// TwinCAT 3 PLC project Types
// Title: Types
// Company: TomasRompotl
// ProjectVersion: 0.0.2
// ProgramVersion: 3.1.4024.0
// libraries:
//   Tc2_Standard, * (Beckhoff Automation GmbH)
//   Tc2_System, * (Beckhoff Automation GmbH)
//   Tc2_Utilities, * (Beckhoff Automation GmbH)
//   Tc3_JsonXml, * (Beckhoff Automation GmbH)
//   Tc3_Module, * (Beckhoff Automation GmbH)
//   Base Interfaces,newest,System
// project tree:
//   Any/ AnyTypeUnion.TcDUT, ToAnyType.TcPOU, IsAnyTypeBinded.TcPOU
//   Binding/ BoolBindingReadOnly.TcPOU, BoolBindable.TcIO (not stored), NotBind.TcPOU (not stored), Bind.TcPOU (not stored)
//   Disposable/ Disposable.TcIO
//   Numbers/ Integer.TcDUT (not stored), Decimal.TcDUT, Positive.TcDUT
//   Queryable/ Queryable.TcIO (not stored)
//   Reflection/ Reflection.TcPOU
//   Values/BooleanExpression/ BooleanOperator.TcDUT (not stored), BooleanExpression.TcPOU
//   Values/BooleanExpression/Functions/ And2.TcPOU, And3.TcPOU (not stored), And4.TcPOU, Or2.TcPOU (not stored), Or3.TcPOU, Or4.TcPOU (not stored), Xor2.TcPOU, Xor3.TcPOU (not stored), Xor4.TcPOU (not stored)
//   Values/ BoolValues.TcGVL (not stored), FalseBoolValue.TcPOU, TrueBoolValue.TcPOU (not stored), BoolValue.TcIO
//   Version/ Global_Version.TcGVL
// real-time tasks:
//   TASK BindingTestTask: cycle T#10ms, priority 20, ADS port 350
//   TASK PlcTask: cycle T#10ms, priority 21, ADS port 351
//   TASK PlcTask1: cycle T#10ms, priority 22, ADS port 352
//   TASK PlcTask2: cycle T#10ms, priority 23, ADS port 353

// ---- Any/AnyTypeUnion.TcDUT
TYPE AnyTypeUnion :
UNION
	BOOL_ : BOOL;
	BIT_ : BIT;
	BYTE_ : BYTE;
	WORD_ : WORD;
	DWORD_ : DWORD;
	LWORD_ : LWORD;
	SINT_ : SINT;
	INT_ : INT;
	DINT_ : DINT;
	LINT_ : LINT;
	USINT_ : USINT;
	UINT_ : UINT;
	UDINT_ : UDINT;
	ULINT_ : ULINT;
	REAL_ : REAL;
	LREAL_ : LREAL;
	STRING_ : T_MaxString;
	TIME_ : TIME;
	DATE_ : DATE;
	DATEANDTIME_ : DATE_AND_TIME;
	TIMEOFDAY_ : TIME_OF_DAY;
	POINTER_ : POINTER TO BYTE;
	LTIME_ : LTIME;
END_UNION
END_TYPE

// ---- Numbers/Decimal.TcDUT
TYPE Decimal : LREAL; END_TYPE

// ---- Numbers/Positive.TcDUT
TYPE Positive : ULINT; END_TYPE

// ---- Version/Global_Version.TcGVL
{attribute 'TcGenerated'}
{attribute 'no-analysis'}
{attribute 'linkalways'}
// This function has been automatically generated from the project information.
VAR_GLOBAL CONSTANT
	{attribute 'const_non_replaced'}
	stLibVersion_Types : ST_LibVersion := (iMajor := 0, iMinor := 0, iBuild := 2, iRevision := 0, nFlags := 0, sVersion := '0.0.2');
END_VAR

// ---- Disposable/Disposable.TcIO
INTERFACE Disposable EXTENDS Queryable

METHOD Dispose
END_METHOD

END_INTERFACE

// ---- Values/BoolValue.TcIO
INTERFACE BoolValue EXTENDS Queryable

{attribute 'monitoring' := 'call'}
PROPERTY Value : BOOL
GET
END_GET
END_PROPERTY

END_INTERFACE

// ---- Any/ToAnyType.TcPOU
FUNCTION ToAnyType : __SYSTEM.AnyType
VAR_INPUT
	object		: ANY;
END_VAR

ToAnyType := object;

END_FUNCTION

// ---- Any/IsAnyTypeBinded.TcPOU
FUNCTION IsAnyTypeBinded : BOOL
VAR_INPUT
	anytype : __SYSTEM.AnyType;
END_VAR

IsAnyTypeBinded := anytype.pValue <> 0 AND anytype.diSize > 0;

END_FUNCTION

// ---- Binding/BoolBindingReadOnly.TcPOU
{attribute 'hide_all_locals'}
{attribute 'enable_dynamic_creation'}
FUNCTION_BLOCK BoolBindingReadOnly IMPLEMENTS BoolBindable
VAR
	ref : REFERENCE TO BOOL;
	_Negate : BOOL;
END_VAR

METHOD Bind
VAR_INPUT
	boolean : REFERENCE TO BOOL;
END_VAR
ref REF= boolean;
END_METHOD

{attribute 'monitoring' := 'call'}
PROPERTY IsBinded : BOOL
GET
IsBinded := __ISVALIDREF(ref);
END_GET
END_PROPERTY

PROPERTY Negate : BOOL
GET
Negate := _Negate;
END_GET
SET
_Negate := Negate;
END_SET
END_PROPERTY

{attribute 'monitoring' := 'call'}
PROPERTY Value : BOOL
GET
Value := ref XOR _Negate;
END_GET
END_PROPERTY

END_FUNCTION_BLOCK

// ---- Reflection/Reflection.TcPOU
{attribute 'hide_all_locals'}
{attribute 'reflection'}
FUNCTION_BLOCK Reflection
VAR
    {attribute 'instance-path'} 
    {attribute 'noinit'} 
    reflectionInstanceName : T_MaxString;
	typeReader : FB_JsonReadWriteDatatype;

	parent : POINTER TO BYTE;
	parentSize : UDINT;

	_InstanceName : T_MaxString;
	_SolutionName : T_MaxString;
	_ProjectName : T_MaxString;
	_ParentName : T_MaxString;
	_Name : T_MaxString;
	
	_ObjectPath : T_MaxString;
	_TypeName : T_MaxString;
END_VAR

METHOD FB_init : BOOL
VAR_INPUT
	bInitRetains : BOOL; // if TRUE, the retain variables are initialized (warm start / cold start)
	bInCopyCode : BOOL;  // if TRUE, the instance afterwards gets moved into the copy code (online change)
	
	parent : POINTER TO BYTE;
	parentSize : UDINT;
END_VAR
THIS^.parent := parent;
THIS^.parentSize := parentSize;

ParseInstanceName();

_ObjectPath := GetNameOfObject();
_TypeName := GetTypeOfObject();
END_METHOD

METHOD PRIVATE GetNameOfObject : T_MaxString
VAR_INPUT
END_VAR
GetNameOfObject := typeReader.GetSymbolNameByAddress(pData := parent, nData := parentSize);
END_METHOD

METHOD PRIVATE GetTypeOfObject : T_MaxString
VAR_INPUT
END_VAR
GetTypeOfObject := typeReader.GetDatatypeNameByAddress(pData := parent, nData := parentSize);
END_METHOD

{attribute 'monitoring' := 'call'}
PROPERTY InstanceName : T_MaxString
GET
InstanceName := _InstanceName;
END_GET
END_PROPERTY

{attribute 'monitoring' := 'call'}
PROPERTY Name : T_MaxString
GET
Name := _Name;
END_GET
END_PROPERTY

{attribute 'monitoring' := 'call'}
PROPERTY ObjectPath : T_MaxString
GET
ObjectPath := _ObjectPath;
END_GET
END_PROPERTY

{attribute 'monitoring' := 'call'}
PROPERTY ParentName : T_MaxString
GET
ParentName := _ParentName;
END_GET
END_PROPERTY

METHOD PRIVATE ParseInstanceName : T_MaxString
VAR
	right : T_MaxString;
END_VAR
VAR CONSTANT
	Dot : STRING(1) := '.';
END_VAR
FindAndSplit(
	pSeparator := ADR(Dot),
	pSrcString := ADR(reflectionInstanceName),
	pLeftString := ADR(_InstanceName),
	nLeftSize := SIZEOF(_InstanceName),
	pRightString := ADR(right),
	nRightSize := SIZEOF(right),
	bSearchFromRight := TRUE
);

FindAndSplit(
	pSeparator := ADR(Dot),
	pSrcString := ADR(_InstanceName),
	pLeftString := ADR(_SolutionName),
	nLeftSize := SIZEOF(_SolutionName),
	pRightString := ADR(right),
	nRightSize := SIZEOF(right),
	bSearchFromRight := FALSE
);

FindAndSplit(
	pSeparator := ADR(Dot),
	pSrcString := ADR(right),
	pLeftString := ADR(_ProjectName),
	nLeftSize := SIZEOF(_ProjectName),
	pRightString := ADR(right),
	nRightSize := SIZEOF(right),
	bSearchFromRight := FALSE
);

FindAndSplit(
	pSeparator := ADR(Dot),
	pSrcString := ADR(right),
	pLeftString := ADR(_ParentName),
	nLeftSize := SIZEOF(_ParentName),
	pRightString := ADR(right),
	nRightSize := SIZEOF(right),
	bSearchFromRight := FALSE
);

_Name := right;
END_METHOD

{attribute 'monitoring' := 'call'}
PROPERTY ProjectName : T_MaxString
GET
ProjectName := _ProjectName;
END_GET
END_PROPERTY

{attribute 'monitoring' := 'call'}
PROPERTY SolutionName : T_MaxString
GET
SolutionName := _SolutionName;
END_GET
END_PROPERTY

{attribute 'monitoring' := 'call'}
PROPERTY TypeName : T_MaxString
GET
TypeName := _TypeName;
END_GET
END_PROPERTY

END_FUNCTION_BLOCK

// ---- Values/BooleanExpression/BooleanExpression.TcPOU
{attribute 'hide_all_locals'}
{attribute 'enable_dynamic_creation'}
FUNCTION_BLOCK BooleanExpression IMPLEMENTS BoolValue
VAR
	operands : ARRAY[0..MaxIndex - 1] OF BoolValue;
	operandCount : INT;
	operator : BooleanOperator;
END_VAR
VAR CONSTANT
	MaxIndex : INT := 4;
END_VAR

METHOD Clear
VAR
	i : INT;
	p : POINTER TO BYTE;
END_VAR
FOR i := 0 TO operandCount - 1 DO
	__QUERYPOINTER(operands[i], p);
	__DELETE(p);
	operands[i] := 0;
END_FOR

operandCount := 0;
END_METHOD

METHOD Op2
VAR_INPUT
	operator : BooleanOperator;
	value1 : BoolValue;
	value2 : BoolValue;
END_VAR
Clear();

THIS^.operator := operator;

operands[0] := value1;
operands[1] := value2;
operandCount := 2;
END_METHOD

METHOD Op3
VAR_INPUT
	operator : BooleanOperator;
	value1 : BoolValue;
	value2 : BoolValue;
	value3 : BoolValue;
END_VAR
Clear();

THIS^.operator := operator;

operands[0] := value1;
operands[1] := value2;
operands[2] := value3;
operandCount := 3;
END_METHOD

METHOD Op4
VAR_INPUT
	operator : BooleanOperator;
	value1 : BoolValue;
	value2 : BoolValue;
	value3 : BoolValue;
	value4 : BoolValue;
END_VAR
Clear();

THIS^.operator := operator;

operands[0] := value1;
operands[1] := value2;
operands[2] := value3;
operands[3] := value4;
operandCount := 4;
END_METHOD

{attribute 'monitoring' := 'call'}
PROPERTY Value : BOOL
GET
VAR
	i : INT;
	result : BOOL;
END_VAR
IF (operandCount = 0) THEN
	RETURN;
END_IF

CASE operator OF
	
	BooleanOperator.ANDop:
		
		result := operands[0].Value;
		FOR i := 1 TO operandCount - 1 DO
			result := result AND operands[i].Value;
		END_FOR	
		
	BooleanOperator.ORop:
		
		result := operands[0].Value;
		FOR i := 1 TO operandCount - 1 DO
			result := result OR operands[i].Value;
		END_FOR	
		
	BooleanOperator.XORop:
		
		result := operands[0].Value;
		FOR i := 1 TO operandCount - 1 DO
			result := result XOR operands[i].Value;
		END_FOR	
		
END_CASE

Value := result;
END_GET
END_PROPERTY

END_FUNCTION_BLOCK

// ---- Values/BooleanExpression/Functions/And2.TcPOU
FUNCTION And2 : BoolValue
VAR_INPUT
	value1 : BoolValue;
	value2 : BoolValue;
END_VAR
VAR
	p : POINTER TO BooleanExpression;
END_VAR

p := __NEW(BooleanExpression);

p^.Op2(
	operator := BooleanOperator.ANDop,
	value1 := value1,
	value2 := value2
);

And2 := p^;

END_FUNCTION

// ---- Values/BooleanExpression/Functions/And4.TcPOU
FUNCTION And4 : BoolValue
VAR_INPUT
	value1 : BoolValue;
	value2 : BoolValue;
	value3 : BoolValue;
	value4 : BoolValue;
END_VAR
VAR
	p : POINTER TO BooleanExpression;
END_VAR

p := __NEW(BooleanExpression);

p^.Op4(
	operator := BooleanOperator.ANDop,
	value1 := value1,
	value2 := value2,
	value3 := value3,
	value4 := value4
);

And4 := p^;

END_FUNCTION

// ---- Values/BooleanExpression/Functions/Or3.TcPOU
FUNCTION Or3 : BoolValue
VAR_INPUT
	value1 : BoolValue;
	value2 : BoolValue;
	value3 : BoolValue;
END_VAR
VAR
	p : POINTER TO BooleanExpression;
END_VAR

p := __NEW(BooleanExpression);

p^.Op3(
	operator := BooleanOperator.ORop,
	value1 := value1,
	value2 := value2,
	value3 := value3
);

Or3 := p^;

END_FUNCTION

// ---- Values/BooleanExpression/Functions/Xor2.TcPOU
FUNCTION Xor2 : BoolValue
VAR_INPUT
	value1 : BoolValue;
	value2 : BoolValue;
END_VAR
VAR
	p : POINTER TO BooleanExpression;
END_VAR

p := __NEW(BooleanExpression);

p^.Op2(
	operator := BooleanOperator.XORop,
	value1 := value1,
	value2 := value2
);

Xor2 := p^;

END_FUNCTION

// ---- Values/FalseBoolValue.TcPOU
FUNCTION_BLOCK FalseBoolValue IMPLEMENTS BoolValue
VAR
END_VAR

{attribute 'monitoring' := 'call'}
PROPERTY Value : BOOL
GET
Value := FALSE;
END_GET
END_PROPERTY

END_FUNCTION_BLOCK
